(* CODESYS project Utils.library
   Company: _
   DefaultNamespace: Utils
   Title: Utils
   Placeholder: _Utils
   Author: Krystian Lis et al.
   Description: Various utilities
   Version: 1.0.0

Project tree, tasks and I/O mapping:
  libraries: Results, * (_); Tc2_Standard, * (Beckhoff Automation GmbH); Tc2_System, * (Beckhoff Automation GmbH)
  Color/
    Itf/
      interface I_RgbColor: Alpha, Blue, Clone, Green, Raw, Red, Set
    data type Color
    function block RgbColor [ST]: Alpha, Blue, Clone, FB_init, Green, Raw, Red, Set
  Time/
    function GetSysTime [ST]
    function Random [ST]
*)

// Color/Color
TYPE Color : DWORD; END_TYPE

// Color/Itf/I_RgbColor
INTERFACE I_RgbColor

PROPERTY Alpha : BYTE
GET
END_GET
SET
END_SET
END_PROPERTY

PROPERTY Blue : BYTE
GET
END_GET
SET
END_SET
END_PROPERTY

METHOD Clone
VAR_INPUT
	iColor	: I_RgbColor;
END_VAR
END_METHOD

PROPERTY Green : BYTE
GET
END_GET
SET
END_SET
END_PROPERTY

PROPERTY Raw : Color
GET
END_GET
SET
END_SET
END_PROPERTY

PROPERTY Red : BYTE
GET
END_GET
SET
END_SET
END_PROPERTY

METHOD Set
VAR_INPUT
	nRed: USINT;
	nGreen: USINT;
	nBlue: USINT;
	nAlpha: USINT;
END_VAR
END_METHOD

END_INTERFACE

// Color/RgbColor
FUNCTION_BLOCK RgbColor IMPLEMENTS I_RgbColor
VAR
	_r: BYTE;
	_g: BYTE;
	_b: BYTE;
	_a: BYTE;
END_VAR

PROPERTY Alpha : BYTE
GET
Alpha := _a;
END_GET
SET
_a := Alpha;
END_SET
END_PROPERTY

PROPERTY Blue : BYTE
GET
Blue := _b;
END_GET
SET
_b := Blue;
END_SET
END_PROPERTY

METHOD Clone
VAR_INPUT
	iColor	: I_RgbColor;
END_VAR
IF iColor = 0 THEN
	RETURN;
END_IF

_r := iColor.Red;
_b := iColor.Blue;
_g := iColor.Green;
_a := iColor.Alpha;
END_METHOD

METHOD FB_init : BOOL
VAR_INPUT
	bInitRetains : BOOL;
	bInCopyCode : BOOL;
	nRed: USINT;
	nGreen: USINT;
	nBlue: USINT;
	nAlpha: USINT;
END_VAR
Set(nRed, nGreen, nBlue, nAlpha);
END_METHOD

PROPERTY Green : BYTE
GET
Green := _g;
END_GET
SET
_g := Green;
END_SET
END_PROPERTY

PROPERTY Raw : Color
GET
Raw := 	USINT_TO_UDINT(_b) OR
			SHL(USINT_TO_UDINT(_g), 8) OR
			SHL(USINT_TO_UDINT(_r), 16) OR
			SHL(USINT_TO_UDINT(_a), 24);
END_GET
SET
_b := UDINT_TO_USINT(Raw AND 16#FF);
_g := UDINT_TO_USINT(SHR(Raw, 8) AND 16#FF);
_r := UDINT_TO_USINT(SHR(Raw, 16) AND 16#FF);
_a := UDINT_TO_USINT(SHR(Raw, 24) AND 16#FF);
END_SET
END_PROPERTY

PROPERTY Red : BYTE
GET
Red := _r;
END_GET
SET
_r := Red;
END_SET
END_PROPERTY

METHOD Set
VAR_INPUT
	nRed: USINT;
	nGreen: USINT;
	nBlue: USINT;
	nAlpha: USINT;
END_VAR
_r := nRed;
_g := nGreen;
_b := nBlue;
_a := nAlpha;
END_METHOD

END_FUNCTION_BLOCK

// Time/GetSysTime
FUNCTION GetSysTime : ULINT
VAR_INPUT
END_VAR
VAR
END_VAR

GetSysTime := Tc2_System.F_GetSystemTime() - 11644473600000000000;

END_FUNCTION

// Time/Random
FUNCTION Random : LREAL
VAR_STAT
	_nSeed		: INT;
END_VAR
VAR
	_drand		: Tc2_System.DRAND;
END_VAR

_drand(seed := (_nSeed := _nSeed + 1), Num => Random);

END_FUNCTION
